// TwinCAT 3 PLC project TempModel_Fast
// ProgramVersion: 3.1.4026.22
// libraries:
//   Tc2_Standard, * (Beckhoff Automation GmbH)
//   Tc2_System, * (Beckhoff Automation GmbH)
//   Tc3_Module, * (Beckhoff Automation GmbH)
// project tree:
//   GVLs/ GVL_238211770.TcGVL
//   / PlcTask.TcTTO (not stored)
//   POUs/ MAIN.TcPOU, Temp_Model0.TcPOU
// (motion and I/O tree: see PLC project lf_system_plc)
// real-time tasks:
//   TASK PlcTask: cycle T#10ms, priority 21, ADS port 350
//   TASK PlcTask1: cycle T#10ms, priority 22, ADS port 351
//   TASK PlcTask2: cycle T#10ms, priority 20, ADS port 352
//   TASK PlcTask3: cycle T#10ms, priority 23, ADS port 353
// variable links:

// ---- GVLs/GVL_238211770.TcGVL
VAR_GLOBAL CONSTANT
	SS_INITIALIZE: SINT := 0;
	SS_STEP: SINT := 1;
END_VAR

// ---- POUs/MAIN.TcPOU
PROGRAM MAIN
VAR
	fbTempModel : Temp_Model0;
	
	iVolt AT%I* : UINT;
	
	iTempSens1 AT%Q* : UINT;
	iTempSens2 AT%Q* : UINT;
	
END_VAR


fbTempModel(ssMethodType:= , iVolt_U:= iVolt , iTemp1_Y=> iTempSens1, iTemp2_Y=> iTempSens2 );
fbTempModel.ssMethodType := 1;

END_PROGRAM

// ---- POUs/Temp_Model0.TcPOU
FUNCTION_BLOCK Temp_Model0
VAR_INPUT
	ssMethodType: SINT;
	iVolt_U: UINT;
END_VAR
VAR_OUTPUT
	iTemp1_Y: UINT;
	iTemp2_Y: UINT;
END_VAR
VAR
	rtb_Gain1: LREAL;
	rtb_Add1: LREAL;
	i: DINT;
	b_counter: DINT;
	counter_b: DINT;
	DiscreteTransferFcn_states: LREAL;
	Delay_DSTATE: ARRAY[0..227] OF LREAL;
END_VAR



CASE ssMethodType OF
    SS_INITIALIZE: 
        (* SystemInitialize for Atomic SubSystem: '<Root>/Temp_Model' *)
        (* InitializeConditions for Sin: '<S1>/Sine Wave' *)
        b_counter := 0;
        (* End of SystemInitialize for SubSystem: '<Root>/Temp_Model' *)
        (* SystemInitialize for Atomic SubSystem: '<Root>/Temp_Model' *)
        (* InitializeConditions for Delay: '<S1>/Delay' *)

        FOR i := 0 TO 227 DO 
            Delay_DSTATE[i] := 0.0;
        END_FOR;

        (* End of InitializeConditions for Delay: '<S1>/Delay' *)
        

        (* InitializeConditions for Sin: '<S1>/Sine Wave1' *)
        counter_b := 0;
        (* InitializeConditions for DiscreteTransferFcn: '<S1>/Discrete Transfer Fcn' *)
        DiscreteTransferFcn_states := 0.0;
        (* End of SystemInitialize for SubSystem: '<Root>/Temp_Model' *)
    SS_STEP: 
        (* Outputs for Atomic SubSystem: '<Root>/Temp_Model' *)
        (* Sum: '<S1>/Add1' incorporates:
         *  Constant: '<S1>/T_umg1'
         *  Delay: '<S1>/Delay'
         *  Sin: '<S1>/Sine Wave'
         *  Sum: '<S1>/Sum5' *)
        rtb_Add1 := (SIN(((DINT_TO_LREAL(b_counter) * 2.0) * 3.1415926535897931) / 10.0) * 0.2) + (Delay_DSTATE[0] + 25.0);
        (* Sum: '<S1>/Add' incorporates:
         *  Constant: '<S1>/T_umg1'
         *  Delay: '<S1>/Delay'
         *  Sin: '<S1>/Sine Wave1'
         *  Sum: '<S1>/Sum5' *)
        rtb_Gain1 := (SIN(((DINT_TO_LREAL(counter_b) * 2.0) * 3.1415926535897931) / 10.0 + 1.5) * 0.3) + (Delay_DSTATE[0] + 25.0);
        (* Update for Sin: '<S1>/Sine Wave' *)
        b_counter := b_counter + 1;

        IF b_counter = 100 THEN 
            b_counter := 0;
        END_IF;

        (* End of Update for Sin: '<S1>/Sine Wave' *)
        

        (* Update for Delay: '<S1>/Delay' incorporates:
         *  DiscreteTransferFcn: '<S1>/Discrete Transfer Fcn' *)

        FOR i := 0 TO 226 DO 
            Delay_DSTATE[i] := Delay_DSTATE[i + 1];
        END_FOR;

        Delay_DSTATE[227] := 0.01177 * DiscreteTransferFcn_states;
        (* End of Update for Delay: '<S1>/Delay' *)
        

        (* Update for Sin: '<S1>/Sine Wave1' *)
        counter_b := counter_b + 1;

        IF counter_b = 100 THEN 
            counter_b := 0;
        END_IF;

        (* End of Update for Sin: '<S1>/Sine Wave1' *)
        

        (* Update for DiscreteTransferFcn: '<S1>/Discrete Transfer Fcn' incorporates:
         *  DataTypeConversion: '<S1>/Data Type Conversion'
         *  Gain: '<S1>/D//A-Wandler EL4002' *)
        DiscreteTransferFcn_states := (0.00015259254737998596 * UINT_TO_LREAL(iVolt_U)) - (-0.999622285179185 * DiscreteTransferFcn_states);
        (* Outport: '<Root>/iTemp1_Y' incorporates:
         *  DataTypeConversion: '<S1>/Data Type Conversion1'
         *  Gain: '<S1>/Gain' *)
        iTemp1_Y := DINT_TO_UINT(TRUNC(100.0 * rtb_Add1));
        (* Outport: '<Root>/iTemp2_Y' incorporates:
         *  DataTypeConversion: '<S1>/Data Type Conversion2'
         *  Gain: '<S1>/Gain1' *)
        iTemp2_Y := DINT_TO_UINT(TRUNC(100.0 * rtb_Gain1));
        (* End of Outputs for SubSystem: '<Root>/Temp_Model' *)
END_CASE;

END_FUNCTION_BLOCK
